TEXTLIST TextList_zErrorid
  0 = 'no_error'
  1 = 'not_connected'
  2 = 'invalid_state'
  3 = 'homing_error'
  4 = 'cmd_timeout'
  5 = 'TBD_error'
  6 = 'io_error'
  7 = 'unknown_error'
  8 = 'actuator_out_of_pos_range'
  9 = 'actuator_out_of_neg_range'
  10 = 'homing_timeout'
  11 = 'parameter_out_of_range'
  12 = 'trigger_Limit'
  666 = 'emergency_error'
  13 = 'Drive_not_ready_for_operation'
   = ''
END_TEXTLIST

(* stored: Version 1.1.0.1, ProductVersion 3.1.4024.11
   TextList TextList_zErrorid: Id {30bf47e6-f43f-4f2c-ab4d-5968af23c8ec} *)
